// TIA Portal V17 export
// export: Created 2024-06-25T12:57:19.1858124Z, ExportSetting WithDefaults, DisplayName Totally Integrated Automation Portal, DisplayVersion V17 Update 6, DisplayName TIA Portal Openness, DisplayVersion V17 Update 6, DisplayName TIA Portal Version Control Interface, DisplayVersion V17, DisplayName STEP 7 Professional, DisplayVersion V17 Update 6, DisplayName STEP 7 Safety, DisplayVersion V17 Update 6, DisplayName WinCC Advanced, DisplayVersion V17 Update 6
DATA_BLOCK "M"   // DB1
{ S7_Optimized_Access := 'TRUE' }
VERSION : 0.1
// stored: AutoNumber true, DBAccessibleFromOPCUA true, IsOnlyStoredInLoadMemory false, IsRetainMemResEnabled false, IsWriteProtectedInAS false, MemoryReserve 100
   VAR
      F_M1 : Bool;   // M_MODO_OFF
      F_M2 : Bool;   // M_MODO_MAN
      F_M3 : Bool;   // M_MODO_AUTO
      F_M4 : Bool;   // LLAVIN A MAN/LOC
      F_M5 : Bool;   // LLAVIN A AUTO/REM
      F_M6 : Bool;   // LLAVIN A MAN/LOC
      F_M7 : Bool;   // LLAVIN A AUTO/REM
      F_M8 : Bool;
      F_M9 : Bool;   // M_NO_RES_AUTO
      F_M10 : Bool;   // PULSADOR OFF
      F_M11 : Bool;   // PULSADOR MAN
      F_M12 : Bool;   // PULSADOR AUTO
      F_M13 : Bool;   // NO PULSADOR OFF
      F_M14 : Bool;   // NO PULSADOR MAN
      F_M15 : Bool;   // NO PULSADOR AUTO
      F_M16 : Bool;   // RES OFF
      F_M17 : Bool;   // RES MAN
      F_M18 : Bool;   // RES AUTO
      F_M19 : Bool;   // NO RES OFF
      F_M20 : Bool;   // NO RES MAN
   END_VAR
BEGIN
END_DATA_BLOCK
